PROGRAM PRG_Home
VAR
	Lamp01	: OnOffDeviceControl;
	Lamp02	: OnOffDeviceControl;
	
END_VAR


	Lamp01();
	Lamp02();

END_PROGRAM

(* stored: Version 1.1.0.1, ProductVersion 3.1.4024.13
   POU PRG_Home: Id {dbe25c38-c0d1-4648-b8ed-0008a8f3eaf6}, SpecialFunc None *)
